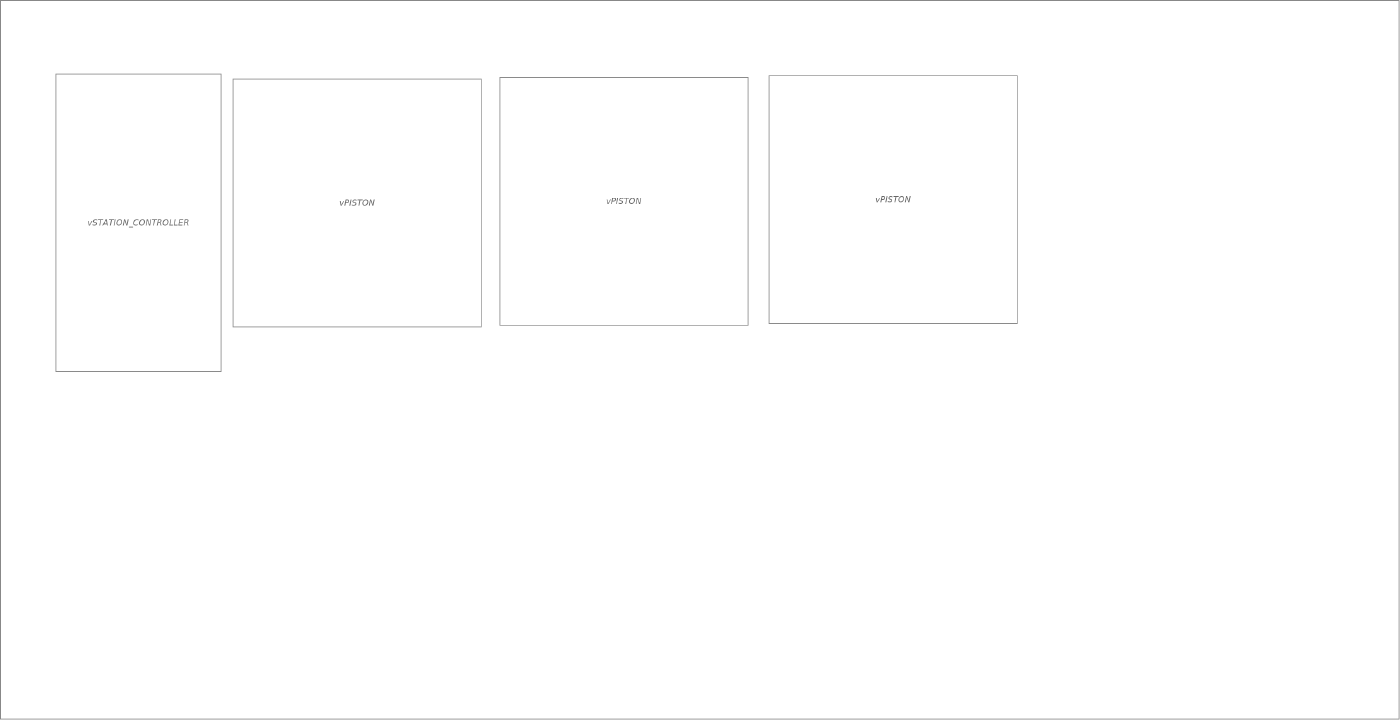
VISUALIZATION vFEEDER  // 1690x870
VAR_IN_OUT
	vFEEDER: FB_FEEDER;
END_VAR
    Frame (281,95 300x300)
        shows vPISTON(PIST1 := vFEEDER.fbPIST1)
    Frame (603,93 300x300)
        shows vPISTON(PIST1 := vFEEDER.fbPIST2)
    Frame (928,91 300x300)
        shows vPISTON(PIST1 := vFEEDER.fbPIST3)
    Frame (67,89 200x360)
        shows vSTATION_CONTROLLER(vSTATION := vFEEDER)
END_VISUALIZATION

(* stored: Version 1.1.0.1, ProductVersion 3.1.4024.12
   Visu vFEEDER: Id {0997d4dd-7eaa-4da0-91a0-77b05d730f48} *)
